Universal Robots URScript: huy.script

def unnamed():
  global _hidden_verificationVariable=0
  set_standard_analog_input_domain(0, 1)
  set_standard_analog_input_domain(1, 1)
  set_tool_analog_input_domain(0, 1)
  set_tool_analog_input_domain(1, 1)
  set_analog_outputdomain(0, 0)
  set_analog_outputdomain(1, 0)
  set_input_actions_to_default()
  set_gravity([0.0, 0.0, 9.82])
  motion_version_set(2)
  tool_wrench_limit_disable()
  set_target_payload(0.000000, [0.000000, 0.000000, 0.000000], [0.000000, 0.000000, 0.000000, 0.000000, 0.000000, 0.000000])
  set_tool_communication(False, 115200, 0, 1, 1.5, 3.5)
  set_tool_output_mode(0)
  set_tool_digital_output_mode(0, 1)
  set_tool_digital_output_mode(1, 1)
  set_tool_voltage(0)
  set_safety_mode_transition_hardness(1)
  set_tcp(p[0.0,0.0,0.0,0.0,0.0,0.0])
  # begin: URCap Installation Node
  #   Source: External Control, 1.0.5, FZI Research Center for Information Technology
  #   Type: External Control
  # end: URCap Installation Node
  step_count_4bec61ef_e10b_4e9b_8a39_236f80bac35b = 0.0
  thread Step_Counter_Thread_e16dbae5_9fb9_4a43_b0d3_1aca2314eaa0():
    while (True):
      step_count_4bec61ef_e10b_4e9b_8a39_236f80bac35b = step_count_4bec61ef_e10b_4e9b_8a39_236f80bac35b + 1.0
      sync()
    end
  end
  run Step_Counter_Thread_e16dbae5_9fb9_4a43_b0d3_1aca2314eaa0()
  while (True):
    $ 2 "Robot Program"
    # begin: URCap Program Node
    #   Source: External Control, 1.0.5, FZI Research Center for Information Technology
    #   Type: External Control
    $ 3 "Control by 192.168.58.10"
popup("The connection to the remote PC at 192.168.58.10:50002 could not be established. Reason: Connection refused (Connection refused)","Receive program failed", False, True, blocking=True)
sync()    # end: URCap Program Node
  end
end
